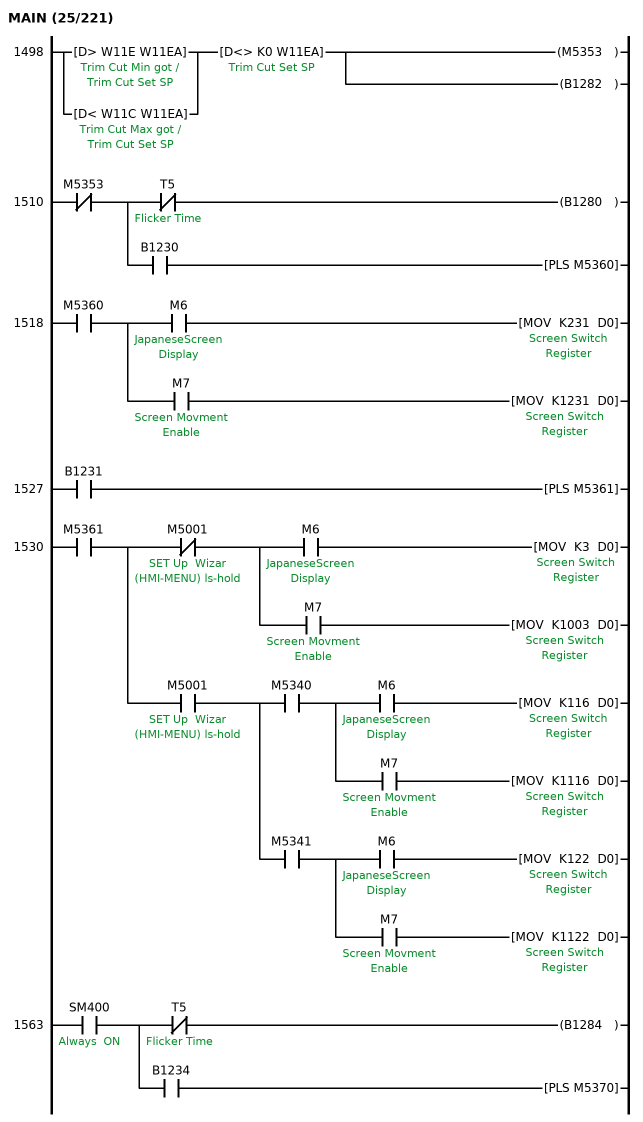
[picture p24: ladder of MAIN, rungs at steps 1498 to 1563]
1498  LDD>    W11E W11EA  ; Trim Cut Min got / Trim Cut Set SP
      ORD<    W11C W11EA  ; Trim Cut Max got / Trim Cut Set SP
      ANDD<>  K0 W11EA  ; Trim Cut Set SP
      OUT     M5353
      OUT     B1282
1510  LDI     M5353
      MPS
      ANI     T5  ; Flicker Time
      OUT     B1280
      MPP
      AND     B1230
      PLS     M5360
1518  LD      M5360
      MPS
      AND     M6  ; JapaneseScreen Display
      MOV     K231 D0
      MPP
      AND     M7  ; Screen Movment Enable
      MOV     K1231 D0
1527  LD      B1231
      PLS     M5361
1530  LD      M5361
      MPS
      ANI     M5001  ; SET Up  Wizar (HMI-MENU) ls-hold
      MPS
      AND     M6  ; JapaneseScreen Display
      MOV     K3 D0
      MPP
      AND     M7  ; Screen Movment Enable
      MOV     K1003 D0
      MPP
      AND     M5001  ; SET Up  Wizar (HMI-MENU) ls-hold
      MPS
      AND     M5340
      MPS
      AND     M6  ; JapaneseScreen Display
      MOV     K116 D0
      MPP
      AND     M7  ; Screen Movment Enable
      MOV     K1116 D0
      MPP
      AND     M5341
      MPS
      AND     M6  ; JapaneseScreen Display
      MOV     K122 D0
      MPP
      AND     M7  ; Screen Movment Enable
      MOV     K1122 D0
1563  LD      SM400  ; Always  ON
      MPS
      ANI     T5  ; Flicker Time
      OUT     B1284
      MPP
      AND     B1234
      PLS     M5370
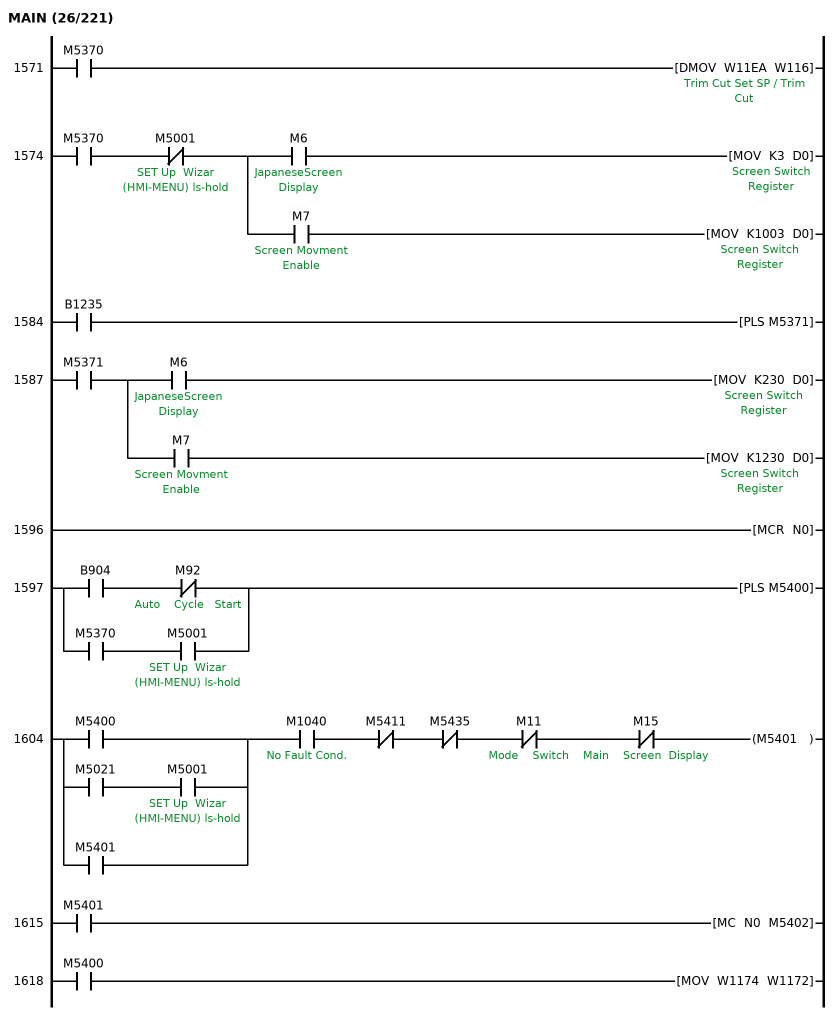
1571  LD      M5370
      DMOV    W11EA W116
1574  LD      M5370
      ANI     M5001  ; SET Up  Wizar (HMI-MENU) ls-hold
      MPS
      AND     M6  ; JapaneseScreen Display
      MOV     K3 D0
      MPP
      AND     M7  ; Screen Movment Enable
      MOV     K1003 D0
1584  LD      B1235
      PLS     M5371
1587  LD      M5371
      MPS
      AND     M6  ; JapaneseScreen Display
      MOV     K230 D0
      MPP
      AND     M7  ; Screen Movment Enable
      MOV     K1230 D0
1596  MCR     N0
1597  LD      B904
      ANI     M92  ; Auto    Cycle   Start
      LD      M5370
      AND     M5001  ; SET Up  Wizar (HMI-MENU) ls-hold
      ORB
      PLS     M5400
1604  LD      M5400
      LD      M5021
      AND     M5001  ; SET Up  Wizar (HMI-MENU) ls-hold
      ORB
      OR      M5401
      AND     M1040  ; No Fault Cond.
      ANI     M5411
      ANI     M5435
      ANI     M11  ; Mode    Switch
      ANI     M15  ; Main    Screen  Display
      OUT     M5401
1615  LD      M5401
      MC      N0 M5402
1618  LD      M5400
      MOV     W1174 W1172
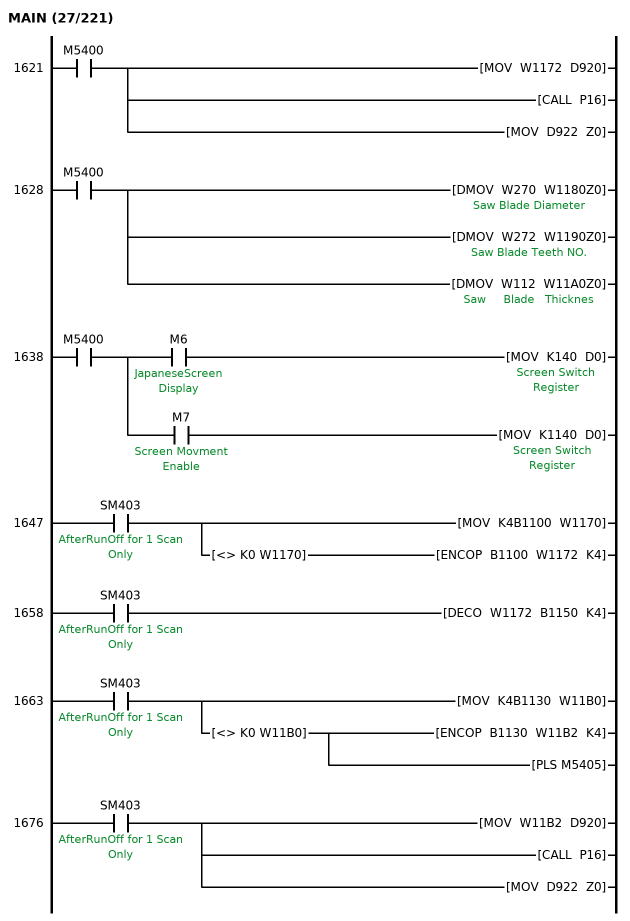
1621  LD      M5400
      MOV     W1172 D920
      CALL    P16
      MOV     D922 Z0
1628  LD      M5400
      DMOV    W270 W1180Z0  ; Saw Blade Diameter
      DMOV    W272 W1190Z0  ; Saw Blade Teeth NO.
      DMOV    W112 W11A0Z0  ; Saw     Blade   Thicknes
1638  LD      M5400
      MPS
      AND     M6  ; JapaneseScreen Display
      MOV     K140 D0
      MPP
      AND     M7  ; Screen Movment Enable
      MOV     K1140 D0
1647  LD      SM403  ; AfterRunOff for 1 Scan  Only
      MOV     K4B1100 W1170
      AND<>   K0 W1170
      ENCOP   B1100 W1172 K4
1658  LD      SM403  ; AfterRunOff for 1 Scan  Only
      DECO    W1172 B1150 K4
1663  LD      SM403  ; AfterRunOff for 1 Scan  Only
      MOV     K4B1130 W11B0
      AND<>   K0 W11B0
      ENCOP   B1130 W11B2 K4
      PLS     M5405
1676  LD      SM403  ; AfterRunOff for 1 Scan  Only
      MOV     W11B2 D920
      CALL    P16
      MOV     D922 Z0
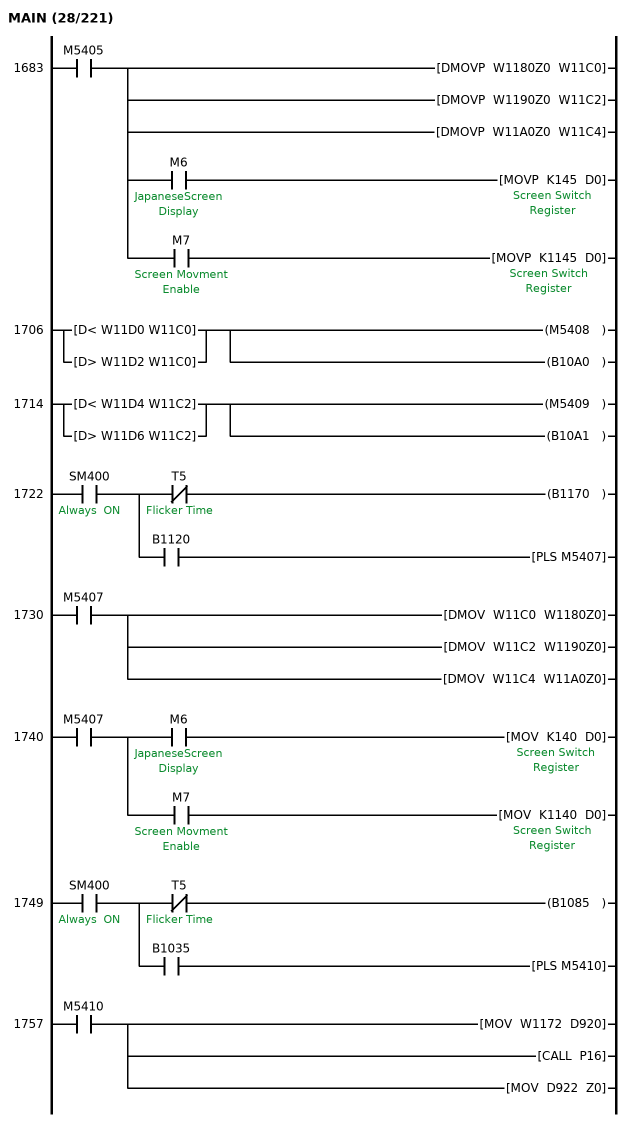
1683  LD      M5405
      DMOVP   W1180Z0 W11C0
      DMOVP   W1190Z0 W11C2
      DMOVP   W11A0Z0 W11C4
      MPS
      AND     M6  ; JapaneseScreen Display
      MOVP    K145 D0
      MPP
      AND     M7  ; Screen Movment Enable
      MOVP    K1145 D0
1706  LDD<    W11D0 W11C0
      ORD>    W11D2 W11C0
      OUT     M5408
      OUT     B10A0
1714  LDD<    W11D4 W11C2
      ORD>    W11D6 W11C2
      OUT     M5409
      OUT     B10A1
1722  LD      SM400  ; Always  ON
      MPS
      ANI     T5  ; Flicker Time
      OUT     B1170
      MPP
      AND     B1120
      PLS     M5407
1730  LD      M5407
      DMOV    W11C0 W1180Z0
      DMOV    W11C2 W1190Z0
      DMOV    W11C4 W11A0Z0
1740  LD      M5407
      MPS
      AND     M6  ; JapaneseScreen Display
      MOV     K140 D0
      MPP
      AND     M7  ; Screen Movment Enable
      MOV     K1140 D0
1749  LD      SM400  ; Always  ON
      MPS
      ANI     T5  ; Flicker Time
      OUT     B1085
      MPP
      AND     B1035
      PLS     M5410
1757  LD      M5410
      MOV     W1172 D920
      CALL    P16
      MOV     D922 Z0
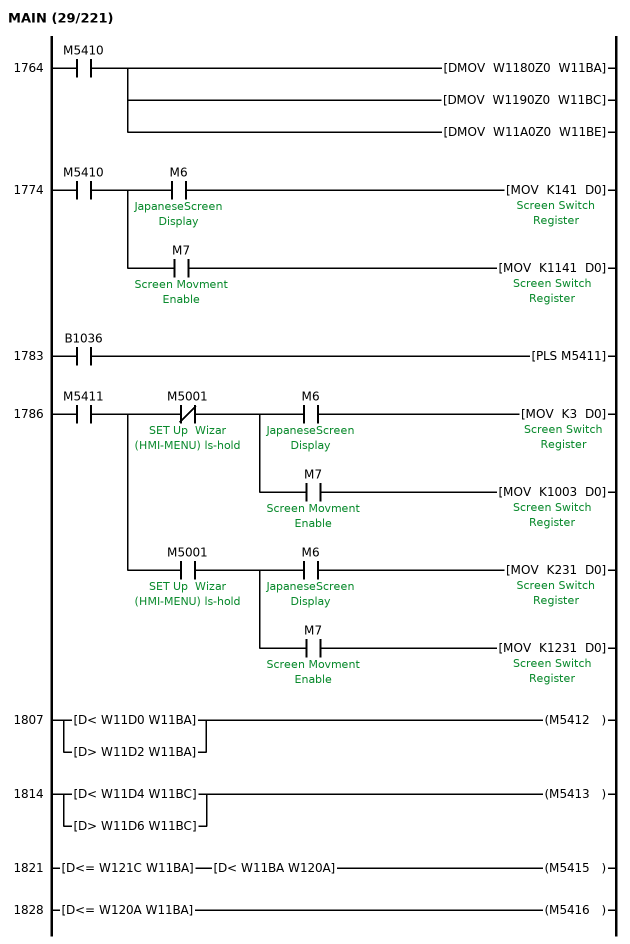
1764  LD      M5410
      DMOV    W1180Z0 W11BA
      DMOV    W1190Z0 W11BC
      DMOV    W11A0Z0 W11BE
1774  LD      M5410
      MPS
      AND     M6  ; JapaneseScreen Display
      MOV     K141 D0
      MPP
      AND     M7  ; Screen Movment Enable
      MOV     K1141 D0
1783  LD      B1036
      PLS     M5411
1786  LD      M5411
      MPS
      ANI     M5001  ; SET Up  Wizar (HMI-MENU) ls-hold
      MPS
      AND     M6  ; JapaneseScreen Display
      MOV     K3 D0
      MPP
      AND     M7  ; Screen Movment Enable
      MOV     K1003 D0
      MPP
      AND     M5001  ; SET Up  Wizar (HMI-MENU) ls-hold
      MPS
      AND     M6  ; JapaneseScreen Display
      MOV     K231 D0
      MPP
      AND     M7  ; Screen Movment Enable
      MOV     K1231 D0
1807  LDD<    W11D0 W11BA
      ORD>    W11D2 W11BA
      OUT     M5412
1814  LDD<    W11D4 W11BC
      ORD>    W11D6 W11BC
      OUT     M5413
1821  LDD<=   W121C W11BA
      ANDD<   W11BA W120A
      OUT     M5415
1828  LDD<=   W120A W11BA
      OUT     M5416
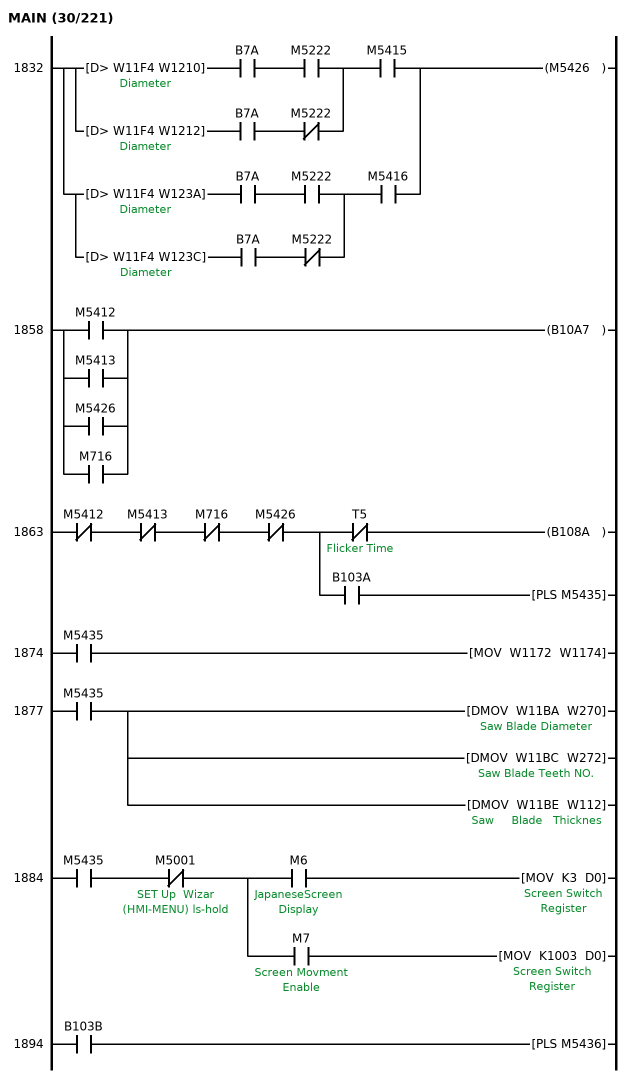
1832  LDD>    W11F4 W1210  ; Diameter
      AND     B7A
      AND     M5222
      LDD>    W11F4 W1212  ; Diameter
      AND     B7A
      ANI     M5222
      ORB
      AND     M5415
      LDD>    W11F4 W123A  ; Diameter
      AND     B7A
      AND     M5222
      LDD>    W11F4 W123C  ; Diameter
      AND     B7A
      ANI     M5222
      ORB
      AND     M5416
      ORB
      OUT     M5426
1858  LD      M5412
      OR      M5413
      OR      M5426
      OR      M716
      OUT     B10A7
1863  LDI     M5412
      ANI     M5413
      ANI     M716
      ANI     M5426
      MPS
      ANI     T5  ; Flicker Time
      OUT     B108A
      MPP
      AND     B103A
      PLS     M5435
1874  LD      M5435
      MOV     W1172 W1174
1877  LD      M5435
      DMOV    W11BA W270
      DMOV    W11BC W272
      DMOV    W11BE W112
1884  LD      M5435
      ANI     M5001  ; SET Up  Wizar (HMI-MENU) ls-hold
      MPS
      AND     M6  ; JapaneseScreen Display
      MOV     K3 D0
      MPP
      AND     M7  ; Screen Movment Enable
      MOV     K1003 D0
1894  LD      B103B
      PLS     M5436
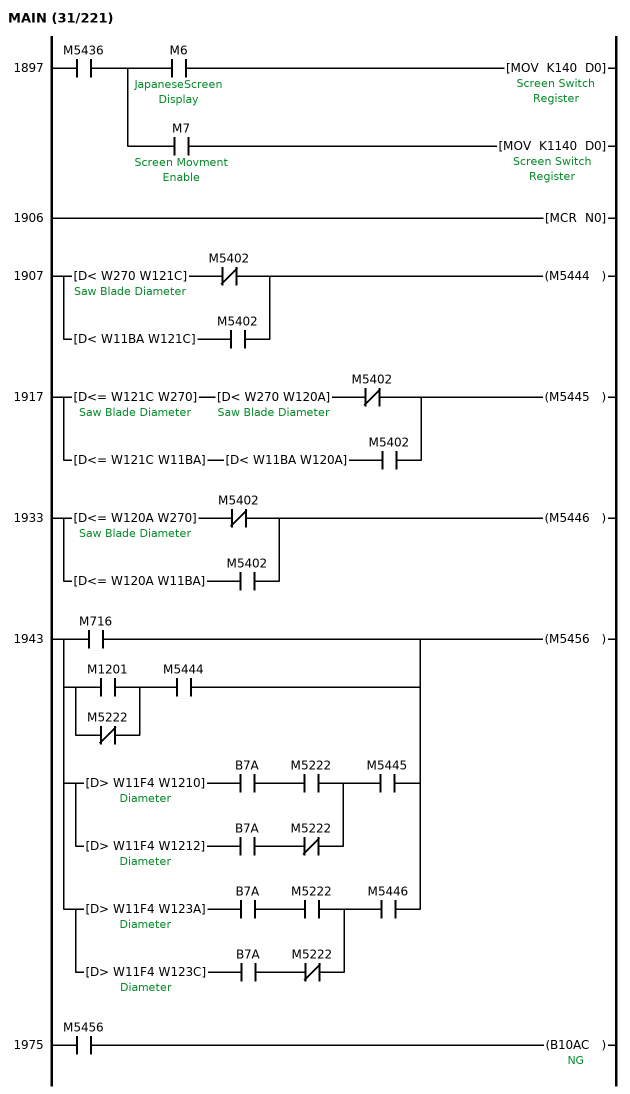
1897  LD      M5436
      MPS
      AND     M6  ; JapaneseScreen Display
      MOV     K140 D0
      MPP
      AND     M7  ; Screen Movment Enable
      MOV     K1140 D0
1906  MCR     N0
1907  LDD<    W270 W121C  ; Saw Blade Diameter
      ANI     M5402
      LDD<    W11BA W121C
      AND     M5402
      ORB
      OUT     M5444
1917  LDD<=   W121C W270  ; Saw Blade Diameter
      ANDD<   W270 W120A  ; Saw Blade Diameter
      ANI     M5402
      LDD<=   W121C W11BA
      ANDD<   W11BA W120A
      AND     M5402
      ORB
      OUT     M5445
1933  LDD<=   W120A W270  ; Saw Blade Diameter
      ANI     M5402
      LDD<=   W120A W11BA
      AND     M5402
      ORB
      OUT     M5446
1943  LD      M716
      LD      M1201
      ORI     M5222
      AND     M5444
      ORB
      LDD>    W11F4 W1210  ; Diameter
      AND     B7A
      AND     M5222
      LDD>    W11F4 W1212  ; Diameter
      AND     B7A
      ANI     M5222
      ORB
      AND     M5445
      ORB
      LDD>    W11F4 W123A  ; Diameter
      AND     B7A
      AND     M5222
      LDD>    W11F4 W123C  ; Diameter
      AND     B7A
      ANI     M5222
      ORB
      AND     M5446
      ORB
      OUT     M5456
1975  LD      M5456
      OUT     B10AC  ; NG
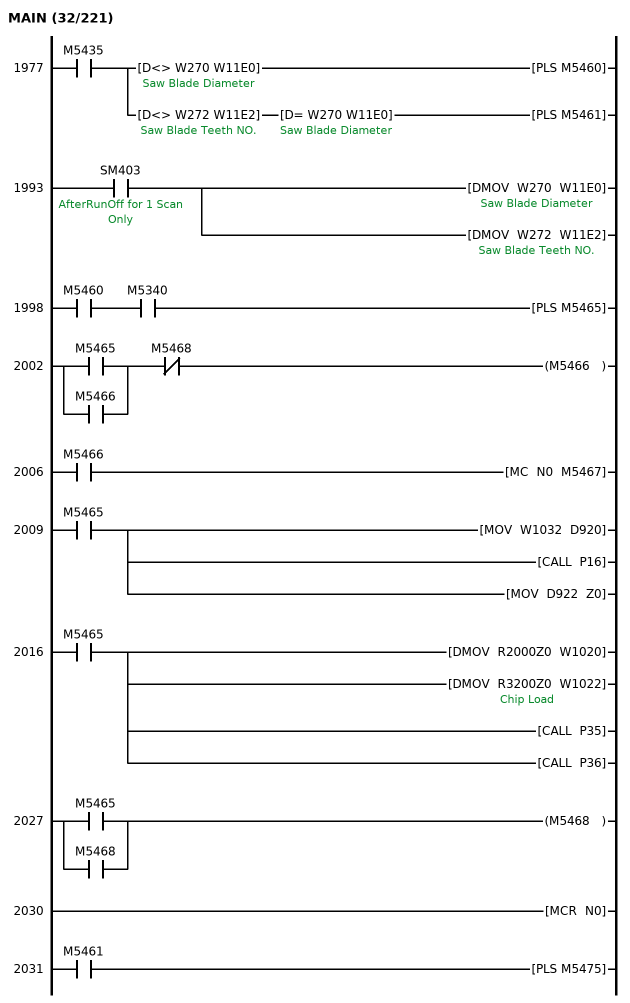
1977  LD      M5435
      MPS
      ANDD<>  W270 W11E0  ; Saw Blade Diameter
      PLS     M5460
      MPP
      ANDD<>  W272 W11E2  ; Saw Blade Teeth NO.
      ANDD=   W270 W11E0  ; Saw Blade Diameter
      PLS     M5461
1993  LD      SM403  ; AfterRunOff for 1 Scan  Only
      DMOV    W270 W11E0
      DMOV    W272 W11E2
1998  LD      M5460
      AND     M5340
      PLS     M5465
2002  LD      M5465
      OR      M5466
      ANI     M5468
      OUT     M5466
2006  LD      M5466
      MC      N0 M5467
2009  LD      M5465
      MOV     W1032 D920
      CALL    P16
      MOV     D922 Z0
2016  LD      M5465
      DMOV    R2000Z0 W1020
      DMOV    R3200Z0 W1022
      CALL    P35
      CALL    P36
2027  LD      M5465
      OR      M5468
      OUT     M5468
2030  MCR     N0
2031  LD      M5461
      PLS     M5475
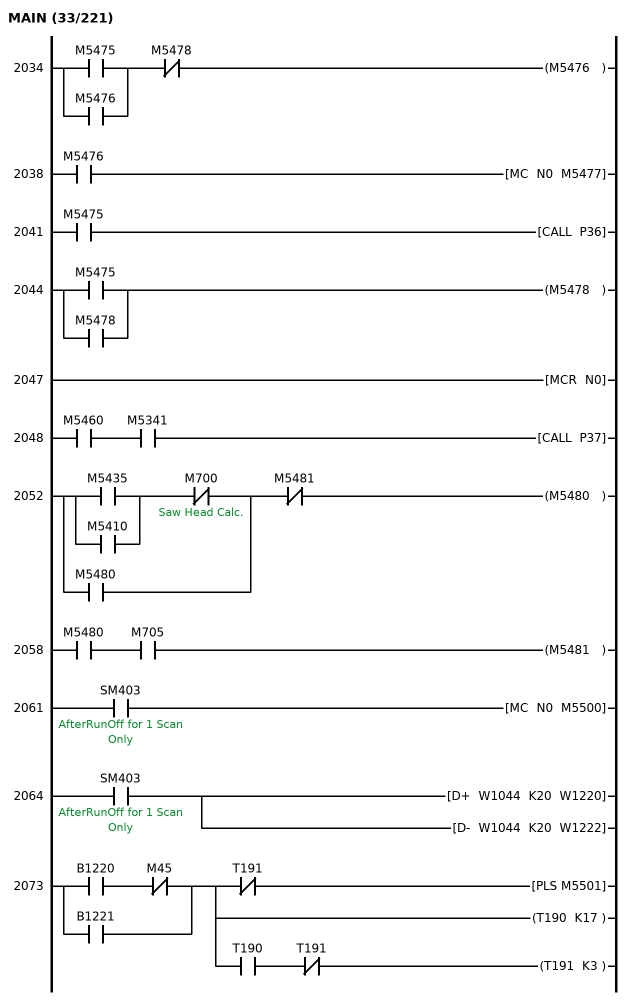
2034  LD      M5475
      OR      M5476
      ANI     M5478
      OUT     M5476
2038  LD      M5476
      MC      N0 M5477
2041  LD      M5475
      CALL    P36
2044  LD      M5475
      OR      M5478
      OUT     M5478
2047  MCR     N0
2048  LD      M5460
      AND     M5341
      CALL    P37
2052  LD      M5435
      OR      M5410
      ANI     M700  ; Saw Head Calc.
      OR      M5480
      ANI     M5481
      OUT     M5480
2058  LD      M5480
      AND     M705
      OUT     M5481
2061  LD      SM403  ; AfterRunOff for 1 Scan  Only
      MC      N0 M5500
2064  LD      SM403  ; AfterRunOff for 1 Scan  Only
      D+      W1044 K20 W1220
      D-      W1044 K20 W1222
2073  LD      B1220
      ANI     M45
      OR      B1221
      MPS
      ANI     T191
      PLS     M5501
      MPP
      OUT     T190 K17
      AND     T190
      ANI     T191
      OUT     T191 K3
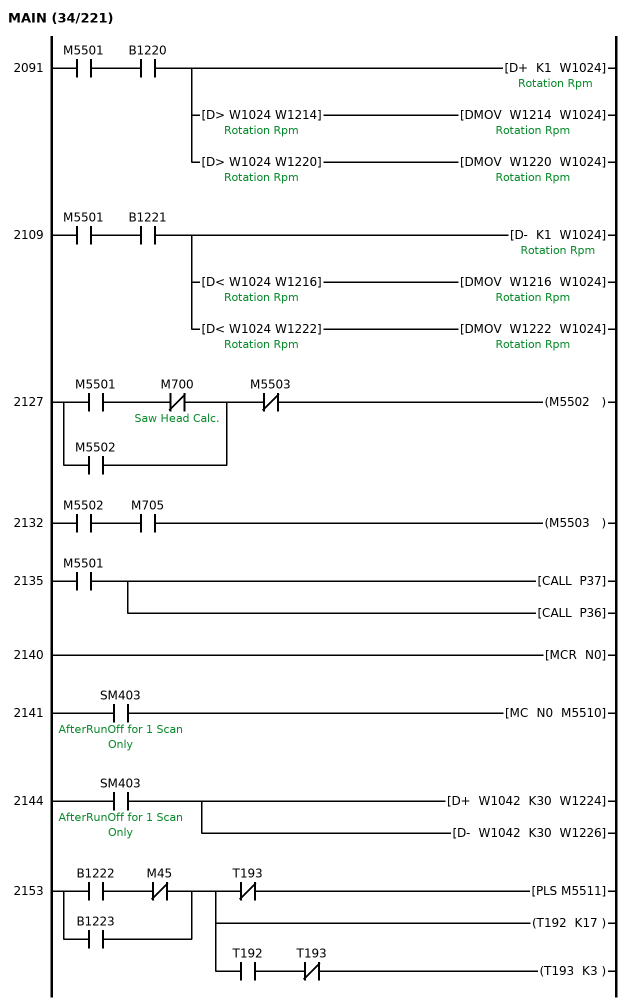
2091  LD      M5501
      AND     B1220
      D+      K1 W1024
      MPS
      ANDD>   W1024 W1214  ; Rotation Rpm
      DMOV    W1214 W1024
      MPP
      ANDD>   W1024 W1220  ; Rotation Rpm
      DMOV    W1220 W1024
2109  LD      M5501
      AND     B1221
      D-      K1 W1024
      MPS
      ANDD<   W1024 W1216  ; Rotation Rpm
      DMOV    W1216 W1024
      MPP
      ANDD<   W1024 W1222  ; Rotation Rpm
      DMOV    W1222 W1024
2127  LD      M5501
      ANI     M700  ; Saw Head Calc.
      OR      M5502
      ANI     M5503
      OUT     M5502
2132  LD      M5502
      AND     M705
      OUT     M5503
2135  LD      M5501
      CALL    P37
      CALL    P36
2140  MCR     N0
2141  LD      SM403  ; AfterRunOff for 1 Scan  Only
      MC      N0 M5510
2144  LD      SM403  ; AfterRunOff for 1 Scan  Only
      D+      W1042 K30 W1224
      D-      W1042 K30 W1226
2153  LD      B1222
      ANI     M45
      OR      B1223
      MPS
      ANI     T193
      PLS     M5511
      MPP
      OUT     T192 K17
      AND     T192
      ANI     T193
      OUT     T193 K3
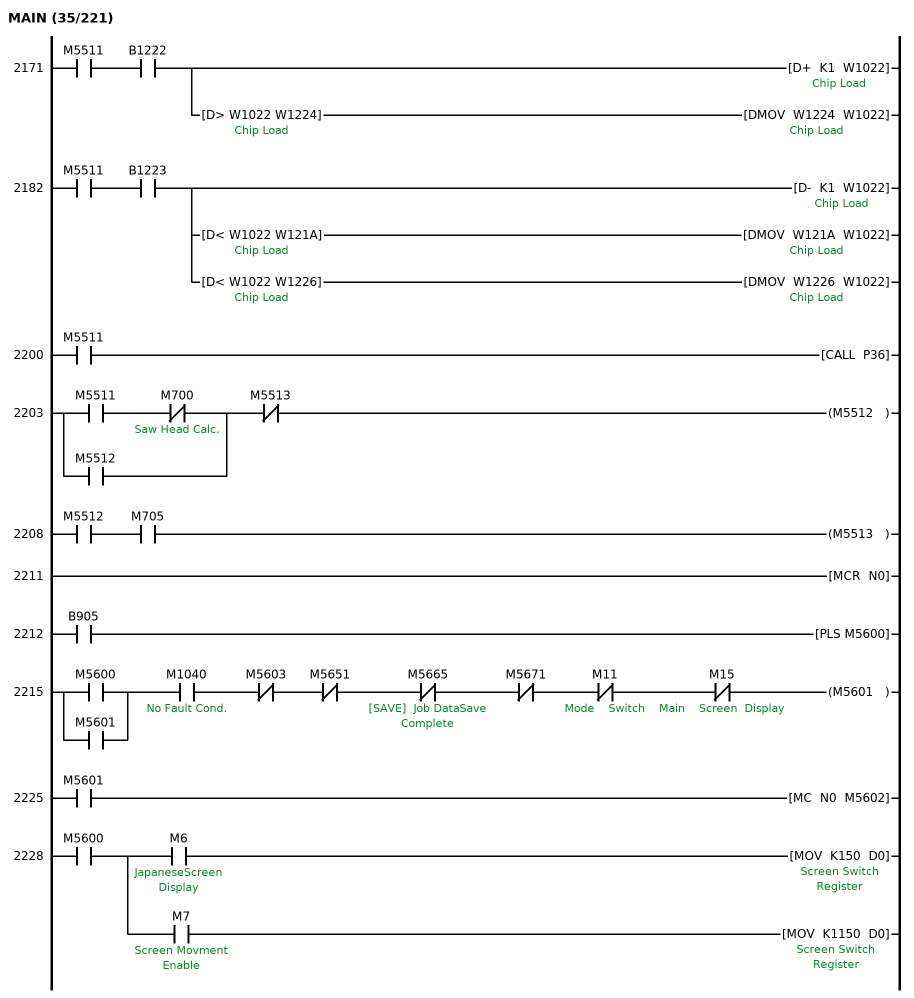
2171  LD      M5511
      AND     B1222
      D+      K1 W1022
      ANDD>   W1022 W1224  ; Chip Load
      DMOV    W1224 W1022
2182  LD      M5511
      AND     B1223
      D-      K1 W1022
      MPS
      ANDD<   W1022 W121A  ; Chip Load
      DMOV    W121A W1022
      MPP
      ANDD<   W1022 W1226  ; Chip Load
      DMOV    W1226 W1022
2200  LD      M5511
      CALL    P36
2203  LD      M5511
      ANI     M700  ; Saw Head Calc.
      OR      M5512
      ANI     M5513
      OUT     M5512
2208  LD      M5512
      AND     M705
      OUT     M5513
2211  MCR     N0
2212  LD      B905
      PLS     M5600
2215  LD      M5600
      OR      M5601
      AND     M1040  ; No Fault Cond.
      ANI     M5603
      ANI     M5651
      ANI     M5665  ; [SAVE]  Job DataSave Complete
      ANI     M5671
      ANI     M11  ; Mode    Switch
      ANI     M15  ; Main    Screen  Display
      OUT     M5601
2225  LD      M5601
      MC      N0 M5602
2228  LD      M5600
      MPS
      AND     M6  ; JapaneseScreen Display
      MOV     K150 D0
      MPP
      AND     M7  ; Screen Movment Enable
      MOV     K1150 D0
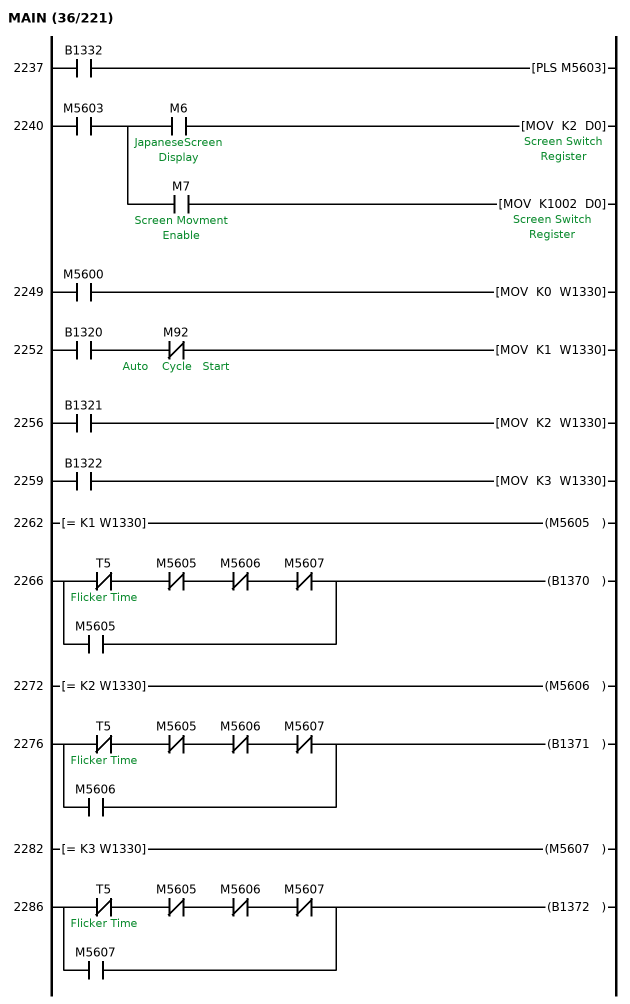
2237  LD      B1332
      PLS     M5603
2240  LD      M5603
      MPS
      AND     M6  ; JapaneseScreen Display
      MOV     K2 D0
      MPP
      AND     M7  ; Screen Movment Enable
      MOV     K1002 D0
2249  LD      M5600
      MOV     K0 W1330
2252  LD      B1320
      ANI     M92  ; Auto    Cycle   Start
      MOV     K1 W1330
2256  LD      B1321
      MOV     K2 W1330
2259  LD      B1322
      MOV     K3 W1330
2262  LD=     K1 W1330
      OUT     M5605
2266  LDI     T5  ; Flicker Time
      ANI     M5605
      ANI     M5606
      ANI     M5607
      OR      M5605
      OUT     B1370
2272  LD=     K2 W1330
      OUT     M5606
2276  LDI     T5  ; Flicker Time
      ANI     M5605
      ANI     M5606
      ANI     M5607
      OR      M5606
      OUT     B1371
2282  LD=     K3 W1330
      OUT     M5607
2286  LDI     T5  ; Flicker Time
      ANI     M5605
      ANI     M5606
      ANI     M5607
      OR      M5607
      OUT     B1372
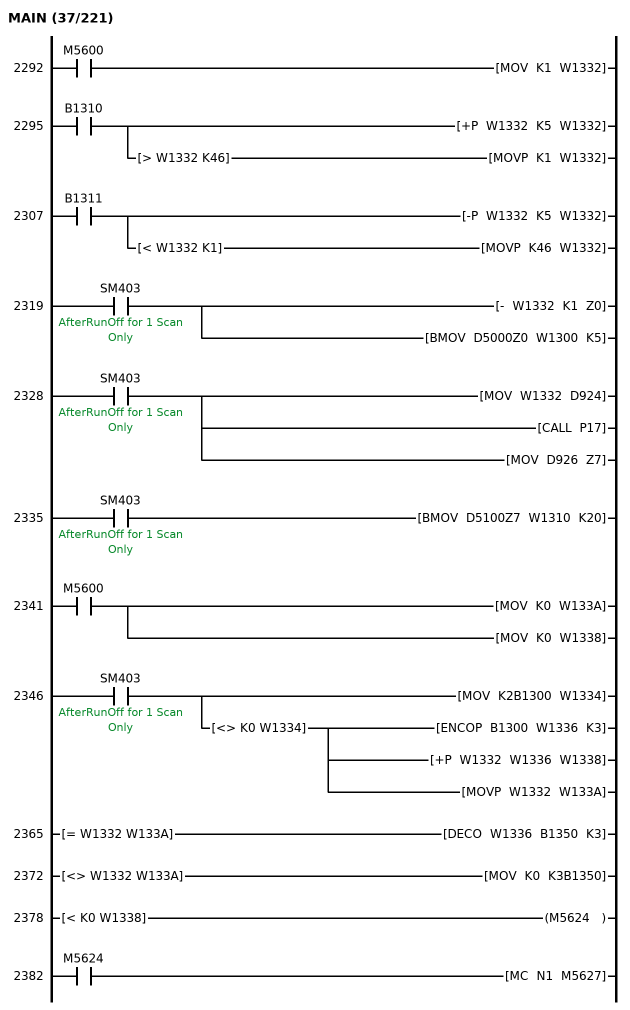
2292  LD      M5600
      MOV     K1 W1332
2295  LD      B1310
      +P      W1332 K5 W1332
      AND>    W1332 K46
      MOVP    K1 W1332
2307  LD      B1311
      -P      W1332 K5 W1332
      AND<    W1332 K1
      MOVP    K46 W1332
2319  LD      SM403  ; AfterRunOff for 1 Scan  Only
      -       W1332 K1 Z0
      BMOV    D5000Z0 W1300 K5
2328  LD      SM403  ; AfterRunOff for 1 Scan  Only
      MOV     W1332 D924
      CALL    P17
      MOV     D926 Z7
2335  LD      SM403  ; AfterRunOff for 1 Scan  Only
      BMOV    D5100Z7 W1310 K20
2341  LD      M5600
      MOV     K0 W133A
      MOV     K0 W1338
2346  LD      SM403  ; AfterRunOff for 1 Scan  Only
      MOV     K2B1300 W1334
      AND<>   K0 W1334
      ENCOP   B1300 W1336 K3
      +P      W1332 W1336 W1338
      MOVP    W1332 W133A
2365  LD=     W1332 W133A
      DECO    W1336 B1350 K3
2372  LD<>    W1332 W133A
      MOV     K0 K3B1350
2378  LD<     K0 W1338
      OUT     M5624
2382  LD      M5624
      MC      N1 M5627
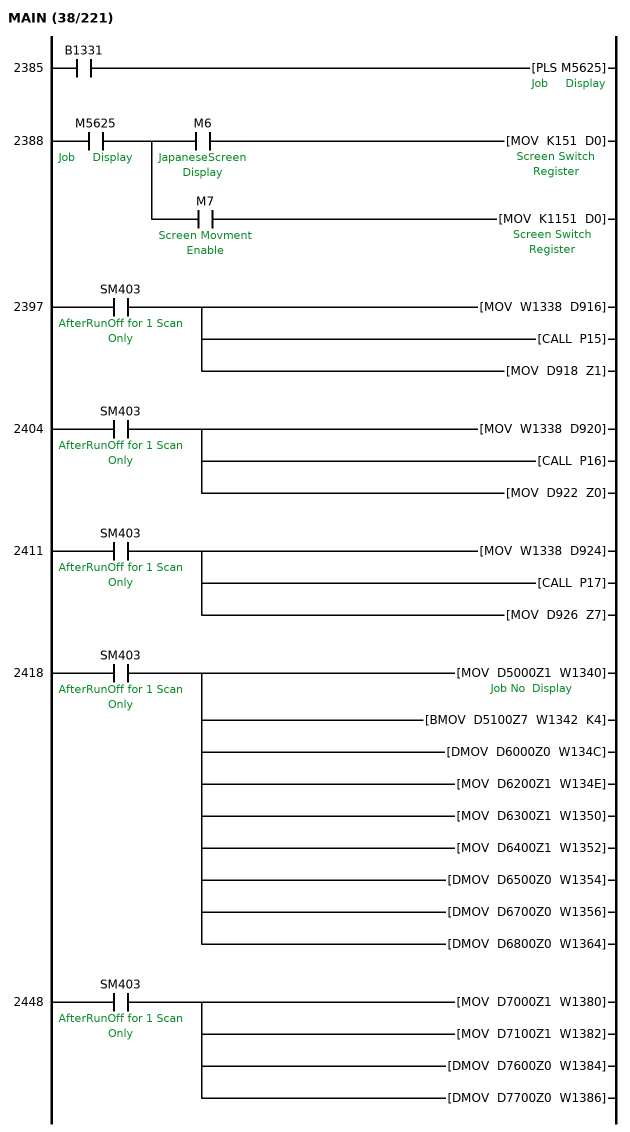
2385  LD      B1331
      PLS     M5625  ; Job     Display
2388  LD      M5625  ; Job     Display
      MPS
      AND     M6  ; JapaneseScreen Display
      MOV     K151 D0
      MPP
      AND     M7  ; Screen Movment Enable
      MOV     K1151 D0
2397  LD      SM403  ; AfterRunOff for 1 Scan  Only
      MOV     W1338 D916
      CALL    P15
      MOV     D918 Z1
2404  LD      SM403  ; AfterRunOff for 1 Scan  Only
      MOV     W1338 D920
      CALL    P16
      MOV     D922 Z0
2411  LD      SM403  ; AfterRunOff for 1 Scan  Only
      MOV     W1338 D924
      CALL    P17
      MOV     D926 Z7
2418  LD      SM403  ; AfterRunOff for 1 Scan  Only
      MOV     D5000Z1 W1340  ; Job No  Display
      BMOV    D5100Z7 W1342 K4
      DMOV    D6000Z0 W134C
      MOV     D6200Z1 W134E
      MOV     D6300Z1 W1350
      MOV     D6400Z1 W1352
      DMOV    D6500Z0 W1354
      DMOV    D6700Z0 W1356
      DMOV    D6800Z0 W1364
2448  LD      SM403  ; AfterRunOff for 1 Scan  Only
      MOV     D7000Z1 W1380
      MOV     D7100Z1 W1382
      DMOV    D7600Z0 W1384
      DMOV    D7700Z0 W1386
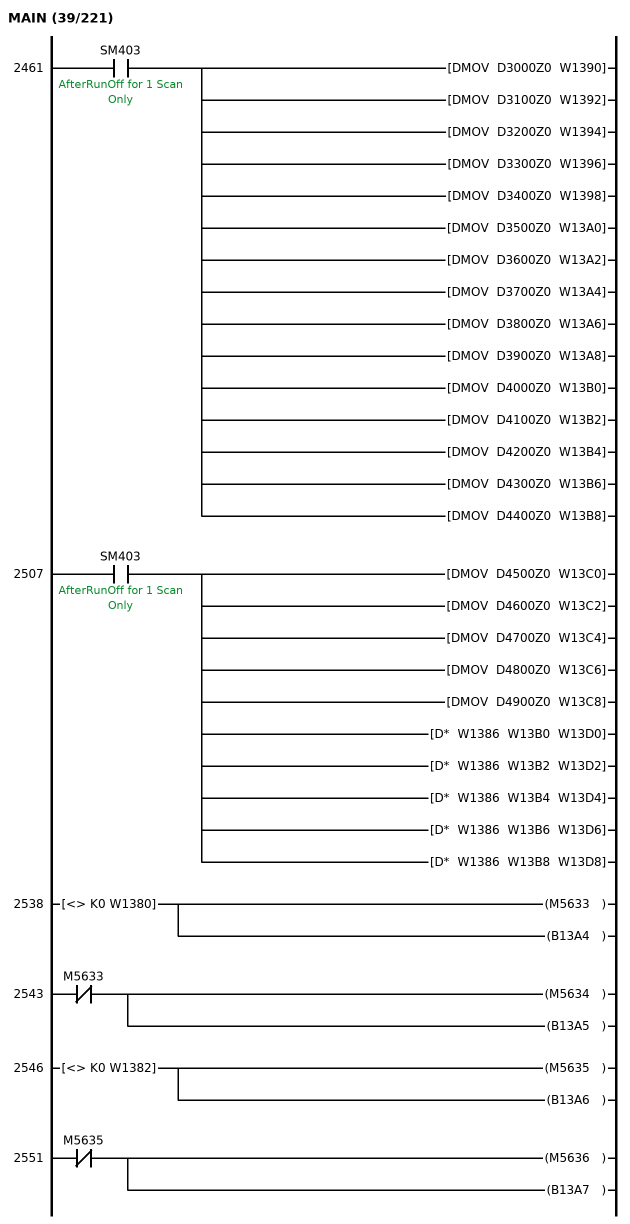
2461  LD      SM403  ; AfterRunOff for 1 Scan  Only
      DMOV    D3000Z0 W1390
      DMOV    D3100Z0 W1392
      DMOV    D3200Z0 W1394
      DMOV    D3300Z0 W1396
      DMOV    D3400Z0 W1398
      DMOV    D3500Z0 W13A0
      DMOV    D3600Z0 W13A2
      DMOV    D3700Z0 W13A4
      DMOV    D3800Z0 W13A6
      DMOV    D3900Z0 W13A8
      DMOV    D4000Z0 W13B0
      DMOV    D4100Z0 W13B2
      DMOV    D4200Z0 W13B4
      DMOV    D4300Z0 W13B6
      DMOV    D4400Z0 W13B8
2507  LD      SM403  ; AfterRunOff for 1 Scan  Only
      DMOV    D4500Z0 W13C0
      DMOV    D4600Z0 W13C2
      DMOV    D4700Z0 W13C4
      DMOV    D4800Z0 W13C6
      DMOV    D4900Z0 W13C8
      D*      W1386 W13B0 W13D0
      D*      W1386 W13B2 W13D2
      D*      W1386 W13B4 W13D4
      D*      W1386 W13B6 W13D6
      D*      W1386 W13B8 W13D8
2538  LD<>    K0 W1380
      OUT     M5633
      OUT     B13A4
2543  LDI     M5633
      OUT     M5634
      OUT     B13A5
2546  LD<>    K0 W1382
      OUT     M5635
      OUT     B13A6
2551  LDI     M5635
      OUT     M5636
      OUT     B13A7
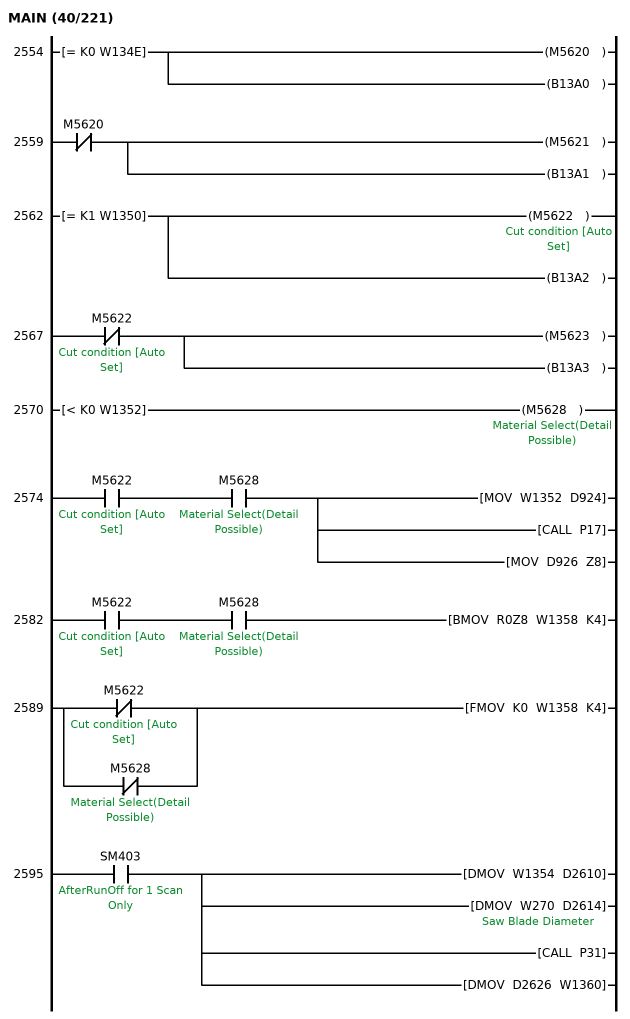
2554  LD=     K0 W134E
      OUT     M5620
      OUT     B13A0
2559  LDI     M5620
      OUT     M5621
      OUT     B13A1
2562  LD=     K1 W1350
      OUT     M5622  ; Cut condition [Auto Set]
      OUT     B13A2
2567  LDI     M5622  ; Cut condition [Auto Set]
      OUT     M5623
      OUT     B13A3
2570  LD<     K0 W1352
      OUT     M5628  ; Material Select(Detail Possible)
2574  LD      M5622  ; Cut condition [Auto Set]
      AND     M5628  ; Material Select(Detail Possible)
      MOV     W1352 D924
      CALL    P17
      MOV     D926 Z8
2582  LD      M5622  ; Cut condition [Auto Set]
      AND     M5628  ; Material Select(Detail Possible)
      BMOV    R0Z8 W1358 K4
2589  LDI     M5622  ; Cut condition [Auto Set]
      ORI     M5628  ; Material Select(Detail Possible)
      FMOV    K0 W1358 K4
2595  LD      SM403  ; AfterRunOff for 1 Scan  Only
      DMOV    W1354 D2610
      DMOV    W270 D2614
      CALL    P31
      DMOV    D2626 W1360
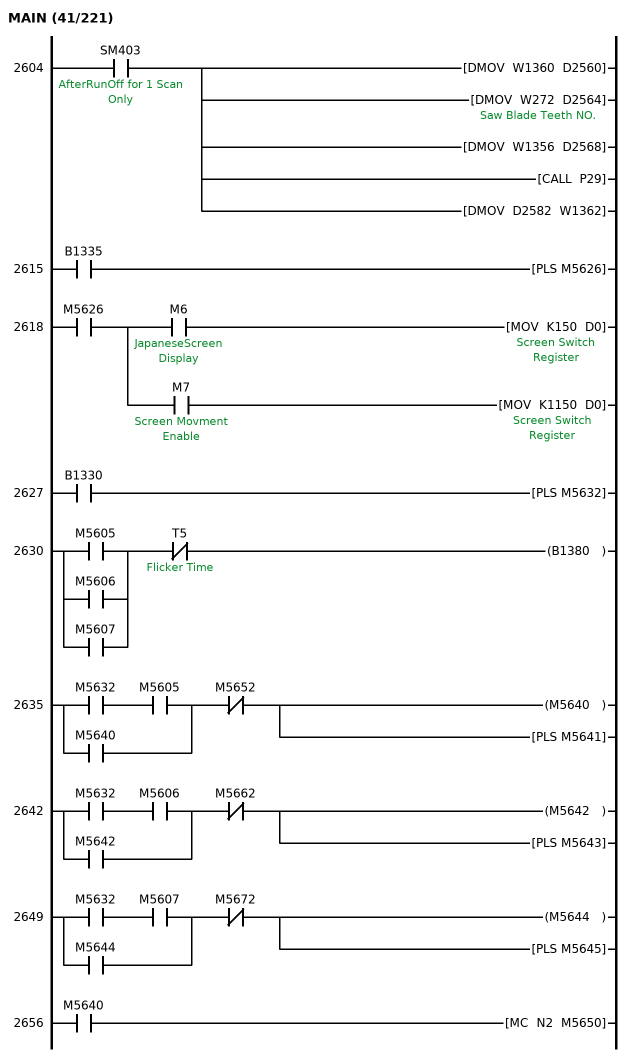
2604  LD      SM403  ; AfterRunOff for 1 Scan  Only
      DMOV    W1360 D2560
      DMOV    W272 D2564
      DMOV    W1356 D2568
      CALL    P29
      DMOV    D2582 W1362
2615  LD      B1335
      PLS     M5626
2618  LD      M5626
      MPS
      AND     M6  ; JapaneseScreen Display
      MOV     K150 D0
      MPP
      AND     M7  ; Screen Movment Enable
      MOV     K1150 D0
2627  LD      B1330
      PLS     M5632
2630  LD      M5605
      OR      M5606
      OR      M5607
      ANI     T5  ; Flicker Time
      OUT     B1380
2635  LD      M5632
      AND     M5605
      OR      M5640
      ANI     M5652
      OUT     M5640
      PLS     M5641
2642  LD      M5632
      AND     M5606
      OR      M5642
      ANI     M5662
      OUT     M5642
      PLS     M5643
2649  LD      M5632
      AND     M5607
      OR      M5644
      ANI     M5672
      OUT     M5644
      PLS     M5645
2656  LD      M5640
      MC      N2 M5650
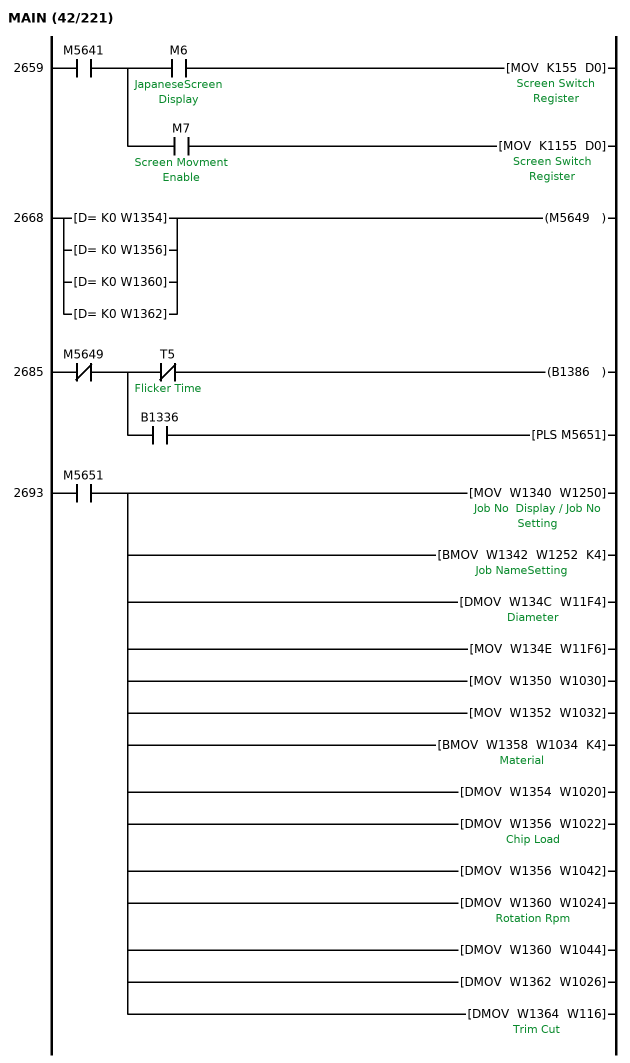
2659  LD      M5641
      MPS
      AND     M6  ; JapaneseScreen Display
      MOV     K155 D0
      MPP
      AND     M7  ; Screen Movment Enable
      MOV     K1155 D0
2668  LDD=    K0 W1354
      ORD=    K0 W1356
      ORD=    K0 W1360
      ORD=    K0 W1362
      OUT     M5649
2685  LDI     M5649
      MPS
      ANI     T5  ; Flicker Time
      OUT     B1386
      MPP
      AND     B1336
      PLS     M5651
2693  LD      M5651
      MOV     W1340 W1250
      BMOV    W1342 W1252 K4
      DMOV    W134C W11F4
      MOV     W134E W11F6
      MOV     W1350 W1030
      MOV     W1352 W1032
      BMOV    W1358 W1034 K4
      DMOV    W1354 W1020
      DMOV    W1356 W1022
      DMOV    W1356 W1042
      DMOV    W1360 W1024
      DMOV    W1360 W1044
      DMOV    W1362 W1026
      DMOV    W1364 W116
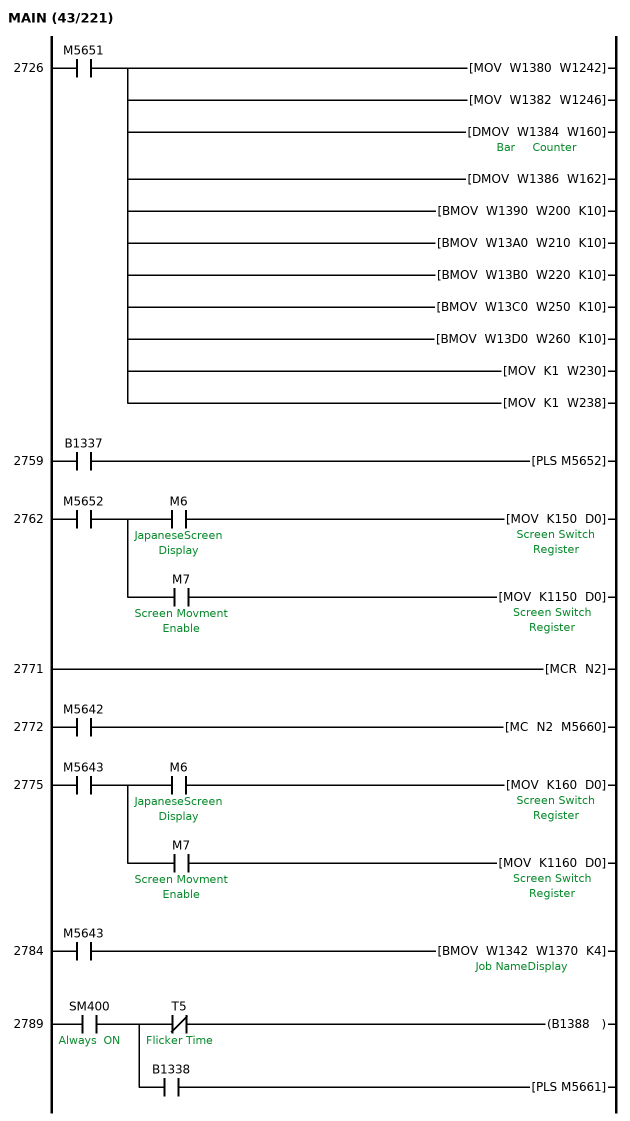
2726  LD      M5651
      MOV     W1380 W1242
      MOV     W1382 W1246
      DMOV    W1384 W160
      DMOV    W1386 W162
      BMOV    W1390 W200 K10
      BMOV    W13A0 W210 K10
      BMOV    W13B0 W220 K10
      BMOV    W13C0 W250 K10
      BMOV    W13D0 W260 K10
      MOV     K1 W230
      MOV     K1 W238
2759  LD      B1337
      PLS     M5652
2762  LD      M5652
      MPS
      AND     M6  ; JapaneseScreen Display
      MOV     K150 D0
      MPP
      AND     M7  ; Screen Movment Enable
      MOV     K1150 D0
2771  MCR     N2
2772  LD      M5642
      MC      N2 M5660
2775  LD      M5643
      MPS
      AND     M6  ; JapaneseScreen Display
      MOV     K160 D0
      MPP
      AND     M7  ; Screen Movment Enable
      MOV     K1160 D0
2784  LD      M5643
      BMOV    W1342 W1370 K4  ; Job NameDisplay
2789  LD      SM400  ; Always  ON
      MPS
      ANI     T5  ; Flicker Time
      OUT     B1388
      MPP
      AND     B1338
      PLS     M5661
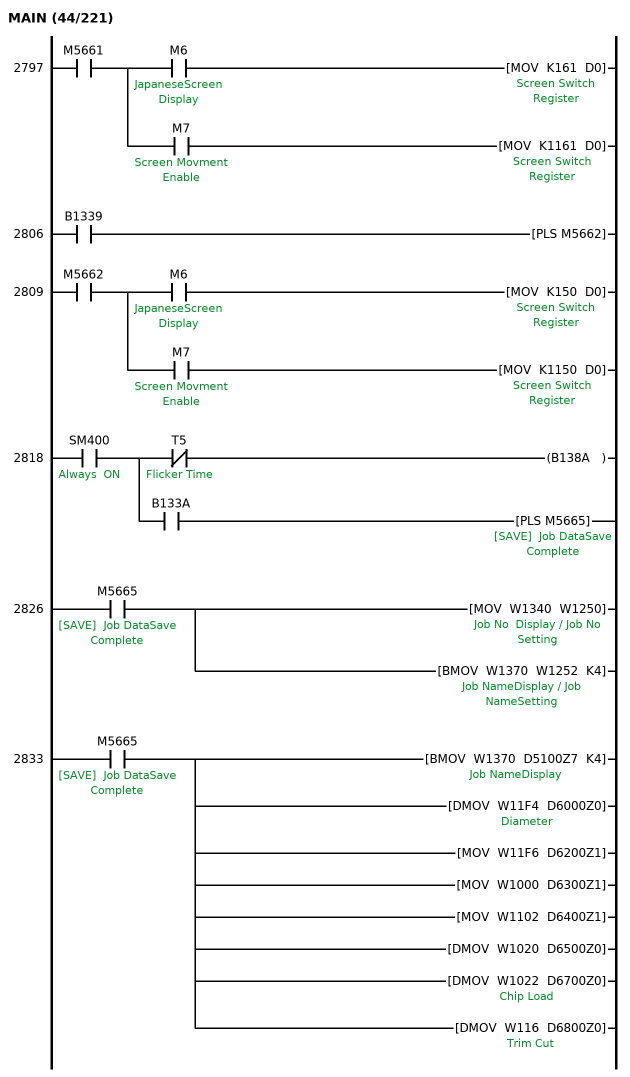
2797  LD      M5661
      MPS
      AND     M6  ; JapaneseScreen Display
      MOV     K161 D0
      MPP
      AND     M7  ; Screen Movment Enable
      MOV     K1161 D0
2806  LD      B1339
      PLS     M5662
2809  LD      M5662
      MPS
      AND     M6  ; JapaneseScreen Display
      MOV     K150 D0
      MPP
      AND     M7  ; Screen Movment Enable
      MOV     K1150 D0
2818  LD      SM400  ; Always  ON
      MPS
      ANI     T5  ; Flicker Time
      OUT     B138A
      MPP
      AND     B133A
      PLS     M5665  ; [SAVE]  Job DataSave Complete
2826  LD      M5665  ; [SAVE]  Job DataSave Complete
      MOV     W1340 W1250
      BMOV    W1370 W1252 K4
2833  LD      M5665  ; [SAVE]  Job DataSave Complete
      BMOV    W1370 D5100Z7 K4
      DMOV    W11F4 D6000Z0
      MOV     W11F6 D6200Z1
      MOV     W1000 D6300Z1
      MOV     W1102 D6400Z1
      DMOV    W1020 D6500Z0
      DMOV    W1022 D6700Z0
      DMOV    W116 D6800Z0
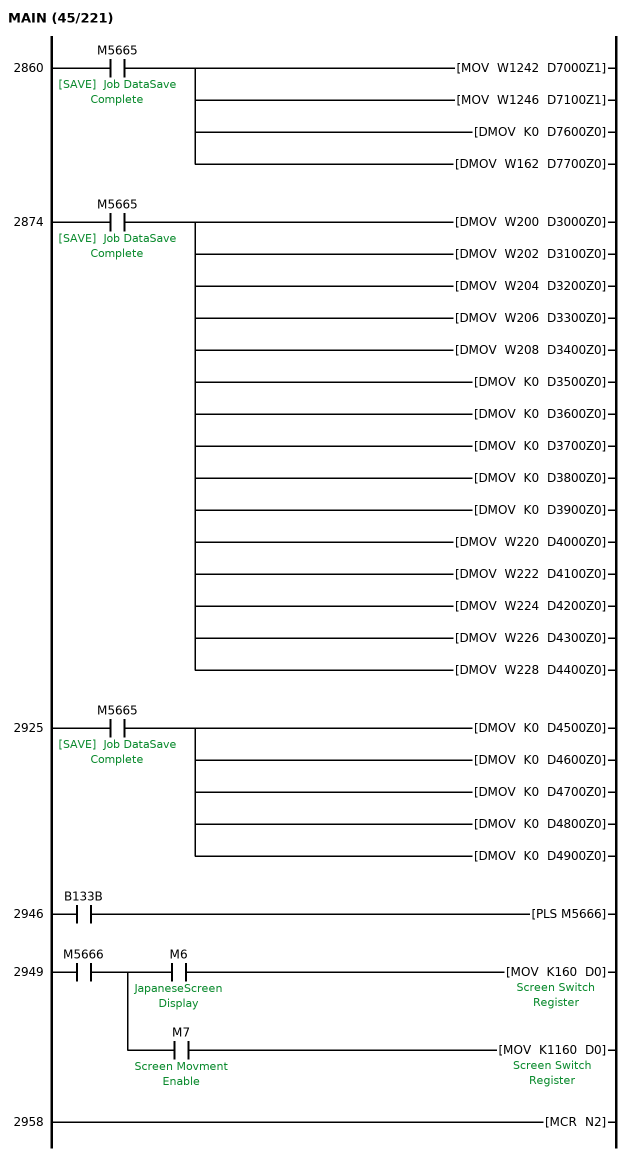
2860  LD      M5665  ; [SAVE]  Job DataSave Complete
      MOV     W1242 D7000Z1
      MOV     W1246 D7100Z1
      DMOV    K0 D7600Z0
      DMOV    W162 D7700Z0
2874  LD      M5665  ; [SAVE]  Job DataSave Complete
      DMOV    W200 D3000Z0
      DMOV    W202 D3100Z0
      DMOV    W204 D3200Z0
      DMOV    W206 D3300Z0
      DMOV    W208 D3400Z0
      DMOV    K0 D3500Z0
      DMOV    K0 D3600Z0
      DMOV    K0 D3700Z0
      DMOV    K0 D3800Z0
      DMOV    K0 D3900Z0
      DMOV    W220 D4000Z0
      DMOV    W222 D4100Z0
      DMOV    W224 D4200Z0
      DMOV    W226 D4300Z0
      DMOV    W228 D4400Z0
2925  LD      M5665  ; [SAVE]  Job DataSave Complete
      DMOV    K0 D4500Z0
      DMOV    K0 D4600Z0
      DMOV    K0 D4700Z0
      DMOV    K0 D4800Z0
      DMOV    K0 D4900Z0
2946  LD      B133B
      PLS     M5666
2949  LD      M5666
      MPS
      AND     M6  ; JapaneseScreen Display
      MOV     K160 D0
      MPP
      AND     M7  ; Screen Movment Enable
      MOV     K1160 D0
2958  MCR     N2
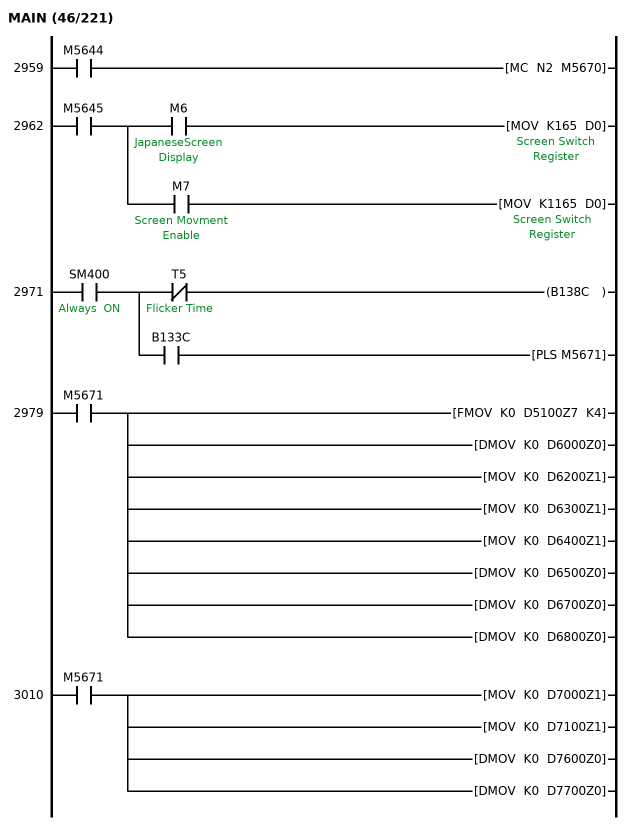
2959  LD      M5644
      MC      N2 M5670
2962  LD      M5645
      MPS
      AND     M6  ; JapaneseScreen Display
      MOV     K165 D0
      MPP
      AND     M7  ; Screen Movment Enable
      MOV     K1165 D0
2971  LD      SM400  ; Always  ON
      MPS
      ANI     T5  ; Flicker Time
      OUT     B138C
      MPP
      AND     B133C
      PLS     M5671
2979  LD      M5671
      FMOV    K0 D5100Z7 K4
      DMOV    K0 D6000Z0
      MOV     K0 D6200Z1
      MOV     K0 D6300Z1
      MOV     K0 D6400Z1
      DMOV    K0 D6500Z0
      DMOV    K0 D6700Z0
      DMOV    K0 D6800Z0
3010  LD      M5671
      MOV     K0 D7000Z1
      MOV     K0 D7100Z1
      DMOV    K0 D7600Z0
      DMOV    K0 D7700Z0
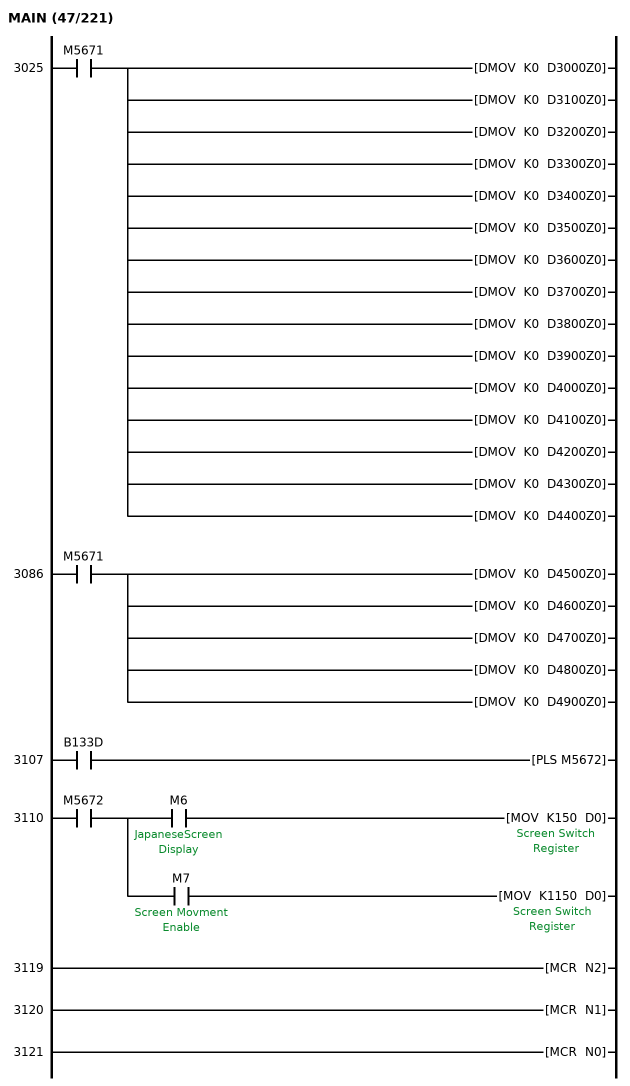
3025  LD      M5671
      DMOV    K0 D3000Z0
      DMOV    K0 D3100Z0
      DMOV    K0 D3200Z0
      DMOV    K0 D3300Z0
      DMOV    K0 D3400Z0
      DMOV    K0 D3500Z0
      DMOV    K0 D3600Z0
      DMOV    K0 D3700Z0
      DMOV    K0 D3800Z0
      DMOV    K0 D3900Z0
      DMOV    K0 D4000Z0
      DMOV    K0 D4100Z0
      DMOV    K0 D4200Z0
      DMOV    K0 D4300Z0
      DMOV    K0 D4400Z0
3086  LD      M5671
      DMOV    K0 D4500Z0
      DMOV    K0 D4600Z0
      DMOV    K0 D4700Z0
      DMOV    K0 D4800Z0
      DMOV    K0 D4900Z0
3107  LD      B133D
      PLS     M5672
3110  LD      M5672
      MPS
      AND     M6  ; JapaneseScreen Display
      MOV     K150 D0
      MPP
      AND     M7  ; Screen Movment Enable
      MOV     K1150 D0
3119  MCR     N2
3120  MCR     N1
3121  MCR     N0
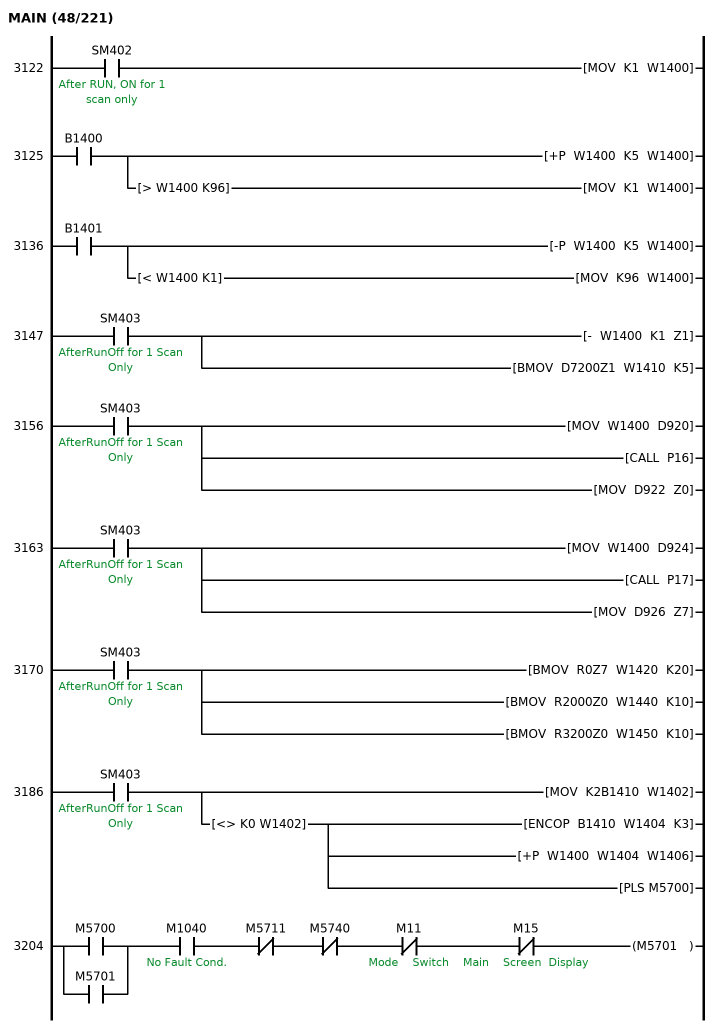
3122  LD      SM402  ; After RUN, ON for 1 scan only
      MOV     K1 W1400
3125  LD      B1400
      +P      W1400 K5 W1400
      AND>    W1400 K96
      MOV     K1 W1400
3136  LD      B1401
      -P      W1400 K5 W1400
      AND<    W1400 K1
      MOV     K96 W1400
3147  LD      SM403  ; AfterRunOff for 1 Scan  Only
      -       W1400 K1 Z1
      BMOV    D7200Z1 W1410 K5
3156  LD      SM403  ; AfterRunOff for 1 Scan  Only
      MOV     W1400 D920
      CALL    P16
      MOV     D922 Z0
3163  LD      SM403  ; AfterRunOff for 1 Scan  Only
      MOV     W1400 D924
      CALL    P17
      MOV     D926 Z7
3170  LD      SM403  ; AfterRunOff for 1 Scan  Only
      BMOV    R0Z7 W1420 K20
      BMOV    R2000Z0 W1440 K10
      BMOV    R3200Z0 W1450 K10
3186  LD      SM403  ; AfterRunOff for 1 Scan  Only
      MOV     K2B1410 W1402
      AND<>   K0 W1402
      ENCOP   B1410 W1404 K3
      +P      W1400 W1404 W1406
      PLS     M5700
3204  LD      M5700
      OR      M5701
      AND     M1040  ; No Fault Cond.
      ANI     M5711
      ANI     M5740
      ANI     M11  ; Mode    Switch
      ANI     M15  ; Main    Screen  Display
      OUT     M5701
